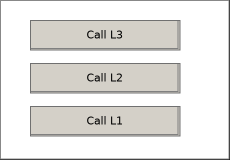
VISUALIZATION CallButtons  // 230x160
VAR_IN_OUT
	L1Call,
	L2Call,
	L3Call:BOOL;
END_VAR
    Rectangle (0,0 230x160)
    Button (30,20 150x30), "Call L3"
        tap L3Call
    Button (30,63 150x30), "Call L2"
        tap L2Call
    Button (30,106 150x30), "Call L1"
        tap L1Call
END_VISUALIZATION

(* stored: Version 1.1.0.1, ProductVersion 3.1.4024.11
   Visu CallButtons: Id {3fed7174-e3e3-4273-a57e-e7e871b88f84} *)
